{attribute 'pack_mode' := '1'}
TYPE ST_TcpTaskBuffer :
STRUCT
	BufferInfo : ARRAY[0..3] OF BYTE;
	TaskData : ST_TcpTask;
END_STRUCT
END_TYPE

(* stored: Version 1.1.0.1, ProductVersion 3.1.4024.12
   DUT ST_TcpTaskBuffer: Id {c26593da-f920-4ee8-b090-2648bc2ab5de} *)
